FUNCTION_BLOCK Test_AddEventHandler_ResizesListWhenListFull EXTENDS TUnitTestBase
VAR_INPUT
END_VAR
VAR_OUTPUT
END_VAR
VAR
    TestEvent : TTestEvent;
    TestEventHandler : TTestEventHandler;
END_VAR

METHOD  Execute
TestEvent
    .ClearEventHandlers()
    .AddEventHandler(TestEventHandler)
    .AddEventHandler(TestEventHandler)
    .AddEventHandler(TestEventHandler)
    .AddEventHandler(TestEventHandler)
    .AddEventHandler(TestEventHandler)  // handler list now full - max handlers = 5
    .AddEventHandler(TestEventHandler); // should trigger an error message
    
Assertion.AssertEquals_UDINT(
    Expected := 6, // 
    Actual   := TestEvent.EventHandlers.Count,
    ObjectName := _TestName,
    VariableName  := 'TestEvent.EventHandlers.Count');

Test_Finished();
END_METHOD

END_FUNCTION_BLOCK

(* stored: Version 1.1.0.1, ProductVersion 3.1.4024.3
   POU Test_AddEventHandler_ResizesListWhenListFull: Id {8d953031-8f81-4063-b7a5-73759d408834}, SpecialFunc None
   Method Execute: Id {51830dec-68d7-422f-af9d-bf9fbef39cee} *)
